// TIA Portal V20 program export: 1 tag tables, 0 data types, 2 data blocks, 4 code blocks (in call order from the OBs), 4 instance data blocks

VAR_GLOBAL   // PLC tag table "默认变量表"
   右顶升V90_Drive_IN AT %I68.0 : "PD_TEL3_IN";
   右顶升V90_Drive_OUT AT %Q68.0 : "PD_TEL3_OUT";
   左顶升IS620F_Drive_IN AT %I86.0 : "PD_TEL3_IN";
   左顶升IS620F_Drive_OUT AT %Q78.0 : "PD_TEL3_OUT";
   System_Byte AT %MB1 : Byte;
   FirstScan AT %M1.0 : Bool;
   DiagStatusUpdate AT %M1.1 : Bool;
   AlwaysTRUE AT %M1.2 : Bool;
   AlwaysFALSE AT %M1.3 : Bool;
   Clock_Byte AT %MB0 : Byte;
   Clock_10Hz AT %M0.0 : Bool;
   Clock_5Hz AT %M0.1 : Bool;
   "Clock_2.5Hz" AT %M0.2 : Bool;
   Clock_2Hz AT %M0.3 : Bool;
   "Clock_1.25Hz" AT %M0.4 : Bool;
   Clock_1Hz AT %M0.5 : Bool;
   "Clock_0.625Hz" AT %M0.6 : Bool;
   "Clock_0.5Hz" AT %M0.7 : Bool;
   右顶升V90控制字 AT %MW2 : Word;
   左顶升IS620F控制字 AT %MW4 : Word;
   左_回原模式 AT %MW6 : Int;
   左_绝对位置 AT %MD8 : Real;
   左_绝对速度 AT %MD12 : Real;
   左_相对位置 AT %MD16 : Real;
   左_相对速度 AT %MD20 : Real;
   左_点动速度 AT %MD24 : Real;
   左顶升IS620F状态字 AT %MW28 : Word;
   左顶升当前位置 AT %MD30 : Real;
   左顶升当前速度 AT %MD34 : Real;
   右顶升V90状态字 AT %MW38 : Word;
   右_回原模式 AT %MW40 : Int;
   右_绝对位置 AT %MD42 : Real;
   右_绝对速度 AT %MD46 : Real;
   右_相对位置 AT %MD50 : Real;
   右_相对速度 AT %MD54 : Real;
   右_点动速度 AT %MD58 : Real;
   右顶升当前位置 AT %MD62 : Real;
   右顶升当前速度 AT %MD66 : Real;
END_VAR

DATA_BLOCK "1200_上传"   // DB2
{ S7_Optimized_Access := 'FALSE' }
   VAR
      位1 : Bool;
      位2 : Bool;
      位3 : Bool;
      位4 : Bool;
      位5 : Bool;
      位6 : Bool;
      位7 : Bool;
      位8 : Bool;
      位9 : Bool;
      位10 : Bool;
      位11 : Bool;
      位12 : Bool;
      位13 : Bool;
      位14 : Bool;
      位15 : Bool;
      位16 : Bool;
      位17 : Bool;
      位18 : Bool;
      位19 : Bool;
      位20 : Bool;
      位21 : Bool;
      位22 : Bool;
      位23 : Bool;
      位24 : Bool;
      位25 : Bool;
      位26 : Bool;
      位27 : Bool;
      位28 : Bool;
      位29 : Bool;
      位30 : Bool;
      整型1 : Int;
      整型2 : Int;
      整型3 : Int;
      整型4 : Int;
      整型5 : Int;
      整型6 : Int;
      整型7 : Int;
      整型8 : Int;
      整型9 : Int;
      整型10 : Int;
      浮点数1 : Real;
      浮点数2 : Real;
      浮点数3 : Real;
      浮点数4 : Real;
      浮点数5 : Real;
      浮点数6 : Real;
      浮点数7 : Real;
      浮点数8 : Real;
      浮点数9 : Real;
      浮点数10 : Real;
      浮点数11 : Real;
      浮点数12 : Real;
      浮点数13 : Real;
      浮点数14 : Real;
      浮点数15 : Real;
      浮点数16 : Real;
      浮点数17 : Real;
      浮点数18 : Real;
      浮点数19 : Real;
   END_VAR
BEGIN
END_DATA_BLOCK

DATA_BLOCK "1200_下载"   // DB1
{ S7_Optimized_Access := 'FALSE' }
   VAR
      位1 : Bool;
      位2 : Bool;
      位3 : Bool;
      位4 : Bool;
      位5 : Bool;
      位6 : Bool;
      位7 : Bool;
      位8 : Bool;
      位9 : Bool;
      位10 : Bool;
      位11 : Bool;
      位12 : Bool;
      位13 : Bool;
      位14 : Bool;
      位15 : Bool;
      位16 : Bool;
      位17 : Bool;
      位18 : Bool;
      位19 : Bool;
      位20 : Bool;
      位21 : Bool;
      位22 : Bool;
      位23 : Bool;
      位24 : Bool;
      位25 : Bool;
      位26 : Bool;
      位27 : Bool;
      位28 : Bool;
      位29 : Bool;
      位30 : Bool;
      整型1 : Int;
      整型2 : Int;
      整型3 : Int;
      整型4 : Int;
      整型5 : Int;
      整型6 : Int;
      整型7 : Int;
      整型8 : Int;
      整型9 : Int;
      整型10 : Int;
      浮点数1 : Real;
      浮点数2 : Real;
      浮点数3 : Real;
      浮点数4 : Real;
      浮点数5 : Real;
      浮点数6 : Real;
      浮点数7 : Real;
      浮点数8 : Real;
      浮点数9 : Real;
      浮点数10 : Real;
      浮点数11 : Real;
      浮点数12 : Real;
      浮点数13 : Real;
      浮点数14 : Real;
      浮点数15 : Real;
      浮点数16 : Real;
      浮点数17 : Real;
      浮点数18 : Real;
      浮点数19 : Real;
   END_VAR
BEGIN
END_DATA_BLOCK

ORGANIZATION_BLOCK "Main"   // OB1, LAD, ProgramCycle
TITLE = "Main Program Sweep (Cycle)"
{ S7_Optimized_Access := 'TRUE' }
// stored: SetENOAutomatically false
   VAR_INPUT
      Initial_Call : Bool;   // Initial call of this OB
      Remanence : Bool;   // =True, if remanent data are available
   END_VAR
   VAR_TEMP
      done : Bool;
      erro : Bool;
      cuowuma : Word;
   END_VAR
BEGIN
END_ORGANIZATION_BLOCK

FUNCTION_BLOCK "定位轴基本控制"   // FB1, LAD
{ S7_Optimized_Access := 'TRUE' }
// stored: MemoryReserve 100, SetENOAutomatically false
   VAR_INPUT
      轴号 : TO_PositioningAxis;
      使能 : Bool;
      回原 : Bool;
      回原模式 : Int;
      绝对定位 : Bool;
      相对定位 : Bool;
      暂停 : Bool;
      复位 : Bool;
      绝对位置 : Real;
      绝对速度 : Real;
      相对位置 : Real;
      相对速度 : Real;
      点动正转 : Bool;
      点动反转 : Bool;
      点动速度 : Real;
   END_VAR
   VAR_OUTPUT
      轴已启用 : Bool;
      使能错误 : Bool;
      回原完成 : Bool;
      回原错误 : Bool;
      绝对定位完成 : Bool;
      绝对定位错误 : Bool;
      相对定位完成 : Bool;
      相对定位错误 : Bool;
      点动中 : Bool;
      点动错误 : Bool;
      当前位置 : Real;
      当前速度 : Real;
   END_VAR
   VAR
      MC_Power_Instance { S7_SetPoint := 'True'} : MC_Power;
      MC_Home_Instance { S7_SetPoint := 'True'} : MC_Home;
      MC_MoveAbsolute_Instance { S7_SetPoint := 'True'} : MC_MoveAbsolute;
      MC_MoveRelative_Instance { S7_SetPoint := 'True'} : MC_MoveRelative;
      MC_Reset_Instance { S7_SetPoint := 'True'} : MC_Reset;
      MC_Halt_Instance { S7_SetPoint := 'True'} : MC_Halt;
      MC_MoveJog_Instance { S7_SetPoint := 'True'} : MC_MoveJog;
   END_VAR
   VAR_TEMP
      复位完成 : Bool;
      复位错误 : Bool;
      暂停完成 : Bool;
      暂停错误 : Bool;
   END_VAR
   VAR_TEMP   // added for the SCL form of the ladder/FBD networks
      _w1 : Bool;
      _w2 : Bool;
      _w3 : Bool;
   END_VAR
BEGIN

REGION Network 1
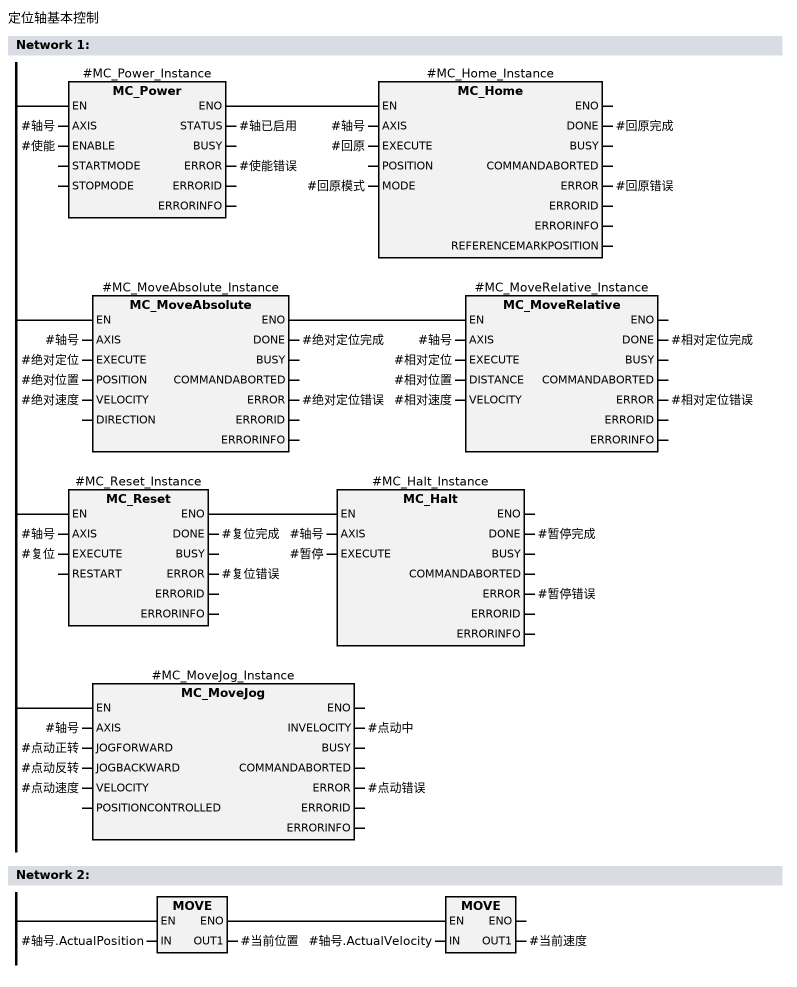
   RUNG wire#powerrail
      #MC_Power_Instance.MC_Power(Axis := #轴号, Enable := #使能, StartMode :=, StopMode :=, Status => #轴已启用, Busy =>, Error => #使能错误, ErrorID =>, ErrorInfo =>)
      #MC_Home_Instance.MC_Home(Axis := #轴号, Execute := #回原, Position :=, Mode := #回原模式, Done => #回原完成, Busy =>, CommandAborted =>, Error => #回原错误, ErrorID =>, ErrorInfo =>, ReferenceMarkPosition =>)
   END_RUNG
   RUNG wire#powerrail
      #MC_MoveAbsolute_Instance.MC_MoveAbsolute(Axis := #轴号, Execute := #绝对定位, Position := #绝对位置, Velocity := #绝对速度, Direction :=, Done => #绝对定位完成, Busy =>, CommandAborted =>, Error => #绝对定位错误, ErrorID =>, ErrorInfo =>)
      #MC_MoveRelative_Instance.MC_MoveRelative(Axis := #轴号, Execute := #相对定位, Distance := #相对位置, Velocity := #相对速度, Done => #相对定位完成, Busy =>, CommandAborted =>, Error => #相对定位错误, ErrorID =>, ErrorInfo =>)
   END_RUNG
   RUNG wire#powerrail
      #MC_Reset_Instance.MC_Reset(Axis := #轴号, Execute := #复位, Restart :=, Done => #复位完成, Busy =>, Error => #复位错误, ErrorID =>, ErrorInfo =>)
      #MC_Halt_Instance.MC_Halt(Axis := #轴号, Execute := #暂停, Done => #暂停完成, Busy =>, CommandAborted =>, Error => #暂停错误, ErrorID =>, ErrorInfo =>)
   END_RUNG
   RUNG wire#powerrail
      #MC_MoveJog_Instance.MC_MoveJog(Axis := #轴号, JogForward := #点动正转, JogBackward := #点动反转, Velocity := #点动速度, PositionControlled :=, InVelocity => #点动中, Busy =>, CommandAborted =>, Error => #点动错误, ErrorID =>, ErrorInfo =>)
   END_RUNG
   // the same network as SCL:
   #MC_Power_Instance(Axis := #轴号, Enable := #使能, Status => #轴已启用, Error => #使能错误, ENO => #_w1);   // MC_Power
   IF #_w1 THEN
       #MC_Home_Instance(Axis := #轴号, Execute := #回原, Mode := #回原模式, Done => #回原完成, Error => #回原错误);   // MC_Home
   END_IF;
   #MC_MoveAbsolute_Instance(Axis := #轴号,   // MC_MoveAbsolute
                           Execute := #绝对定位,
                           Position := #绝对位置,
                           Velocity := #绝对速度,
                           Done => #绝对定位完成,
                           Error => #绝对定位错误,
                           ENO => #_w2);
   IF #_w2 THEN
       #MC_MoveRelative_Instance(Axis := #轴号,   // MC_MoveRelative
                               Execute := #相对定位,
                               Distance := #相对位置,
                               Velocity := #相对速度,
                               Done => #相对定位完成,
                               Error => #相对定位错误);
   END_IF;
   #MC_Reset_Instance(Axis := #轴号, Execute := #复位, Done => #复位完成, Error => #复位错误, ENO => #_w3);   // MC_Reset
   IF #_w3 THEN
       #MC_Halt_Instance(Axis := #轴号, Execute := #暂停, Done => #暂停完成, Error => #暂停错误);   // MC_Halt
   END_IF;
   #MC_MoveJog_Instance(Axis := #轴号,   // MC_MoveJog
                        JogForward := #点动正转,
                        JogBackward := #点动反转,
                        Velocity := #点动速度,
                        InVelocity => #点动中,
                        Error => #点动错误);
END_REGION

REGION Network 2
   RUNG wire#powerrail
      Move(in := #轴号.ActualPosition, out1 => #当前位置)
      Move(in := #轴号.ActualVelocity, out1 => #当前速度)
   END_RUNG
   // the same network as SCL:
   #当前位置 := #轴号.ActualPosition;
   #当前速度 := #轴号.ActualVelocity;
END_REGION
END_FUNCTION_BLOCK

FUNCTION "右顶升伺服" : Void   // FC2, LAD
{ S7_Optimized_Access := 'TRUE' }
// stored: SetENOAutomatically false
BEGIN

REGION Network 1 (SCL)
   "右顶升V90控制字".%X0 := "1200_下载".位9;
   "右顶升V90控制字".%X1 := "1200_下载".位10;
   "右顶升V90控制字".%X2 := "1200_下载".位11;
   "右顶升V90控制字".%X3 := "1200_下载".位12;
   "右顶升V90控制字".%X4 := "1200_下载".位13;
   "右顶升V90控制字".%X5 := "1200_下载".位14;
   "右顶升V90控制字".%X6 := "1200_下载".位15;
   "右顶升V90控制字".%X7 := "1200_下载".位16;

   "右_回原模式" := "1200_下载".整型2;

   "右_绝对位置" := "1200_下载".浮点数6;
   "右_绝对速度" := "1200_下载".浮点数7;
   "右_相对位置" := "1200_下载".浮点数8;
   "右_相对速度" := "1200_下载".浮点数9;
   "右_点动速度" := "1200_下载".浮点数10;
END_REGION

REGION Network 2
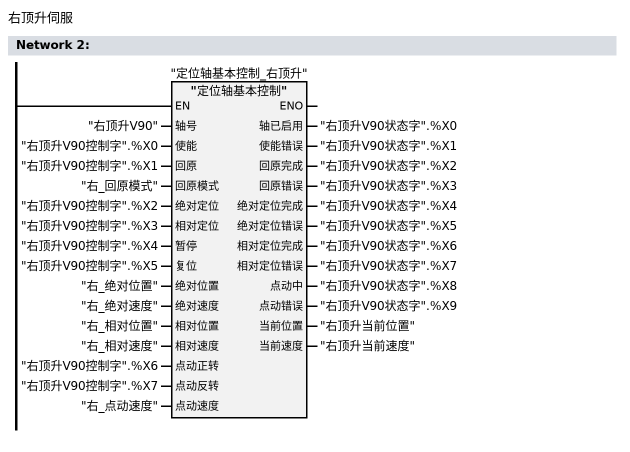
   RUNG wire#powerrail
      "定位轴基本控制_右顶升"(轴号 := "右顶升V90", 使能 := "右顶升V90控制字".%X0, 回原 := "右顶升V90控制字".%X1, 回原模式 := "右_回原模式", 绝对定位 := "右顶升V90控制字".%X2, 相对定位 := "右顶升V90控制字".%X3, 暂停 := "右顶升V90控制字".%X4, 复位 := "右顶升V90控制字".%X5, 绝对位置 := "右_绝对位置", 绝对速度 := "右_绝对速度", 相对位置 := "右_相对位置", 相对速度 := "右_相对速度", 点动正转 := "右顶升V90控制字".%X6, 点动反转 := "右顶升V90控制字".%X7, 点动速度 := "右_点动速度", 轴已启用 => "右顶升V90状态字".%X0, 使能错误 => "右顶升V90状态字".%X1, 回原完成 => "右顶升V90状态字".%X2, 回原错误 => "右顶升V90状态字".%X3, 绝对定位完成 => "右顶升V90状态字".%X4, 绝对定位错误 => "右顶升V90状态字".%X5, 相对定位完成 => "右顶升V90状态字".%X6, 相对定位错误 => "右顶升V90状态字".%X7, 点动中 => "右顶升V90状态字".%X8, 点动错误 => "右顶升V90状态字".%X9, 当前位置 => "右顶升当前位置", 当前速度 => "右顶升当前速度")
   END_RUNG
   // the same network as SCL:
   "定位轴基本控制_右顶升"(轴号 := "右顶升V90",   // "定位轴基本控制"
                 使能 := "右顶升V90控制字".%X0,
                 回原 := "右顶升V90控制字".%X1,
                 回原模式 := "右_回原模式",
                 绝对定位 := "右顶升V90控制字".%X2,
                 相对定位 := "右顶升V90控制字".%X3,
                 暂停 := "右顶升V90控制字".%X4,
                 复位 := "右顶升V90控制字".%X5,
                 绝对位置 := "右_绝对位置",
                 绝对速度 := "右_绝对速度",
                 相对位置 := "右_相对位置",
                 相对速度 := "右_相对速度",
                 点动正转 := "右顶升V90控制字".%X6,
                 点动反转 := "右顶升V90控制字".%X7,
                 点动速度 := "右_点动速度",
                 轴已启用 => "右顶升V90状态字".%X0,
                 使能错误 => "右顶升V90状态字".%X1,
                 回原完成 => "右顶升V90状态字".%X2,
                 回原错误 => "右顶升V90状态字".%X3,
                 绝对定位完成 => "右顶升V90状态字".%X4,
                 绝对定位错误 => "右顶升V90状态字".%X5,
                 相对定位完成 => "右顶升V90状态字".%X6,
                 相对定位错误 => "右顶升V90状态字".%X7,
                 点动中 => "右顶升V90状态字".%X8,
                 点动错误 => "右顶升V90状态字".%X9,
                 当前位置 => "右顶升当前位置",
                 当前速度 => "右顶升当前速度");
END_REGION

REGION Network 3 (SCL)
   "1200_上传".位11 := "右顶升V90状态字".%X0;
   "1200_上传".位12 := "右顶升V90状态字".%X1;
   "1200_上传".位13 := "右顶升V90状态字".%X2;
   "1200_上传".位14 := "右顶升V90状态字".%X3;
   "1200_上传".位15 := "右顶升V90状态字".%X4;
   "1200_上传".位16 := "右顶升V90状态字".%X5;
   "1200_上传".位17 := "右顶升V90状态字".%X6;
   "1200_上传".位18 := "右顶升V90状态字".%X7;
   "1200_上传".位19 := "右顶升V90状态字".%X8;
   "1200_上传".位20 := "右顶升V90状态字".%X9;

   "1200_上传".浮点数3 := "右顶升当前位置";
   "1200_上传".浮点数4 := "右顶升当前速度";
END_REGION
END_FUNCTION

FUNCTION "左顶升伺服" : Void   // FC1, LAD
{ S7_Optimized_Access := 'TRUE' }
// stored: SetENOAutomatically false
BEGIN

REGION Network 1 (SCL)
   "左顶升IS620F控制字".%X0 := "1200_下载".位1;
   "左顶升IS620F控制字".%X1 := "1200_下载".位2;
   "左顶升IS620F控制字".%X2 := "1200_下载".位3;
   "左顶升IS620F控制字".%X3 := "1200_下载".位4;
   "左顶升IS620F控制字".%X4 := "1200_下载".位5;
   "左顶升IS620F控制字".%X5 := "1200_下载".位6;
   "左顶升IS620F控制字".%X6 := "1200_下载".位7;
   "左顶升IS620F控制字".%X7 := "1200_下载".位8;

   "左_回原模式" := "1200_下载".整型1;

   "左_绝对位置" := "1200_下载".浮点数1;
   "左_绝对速度" := "1200_下载".浮点数2;
   "左_相对位置" := "1200_下载".浮点数3;
   "左_相对速度" := "1200_下载".浮点数4;
   "左_点动速度" := "1200_下载".浮点数5;
END_REGION

REGION Network 2
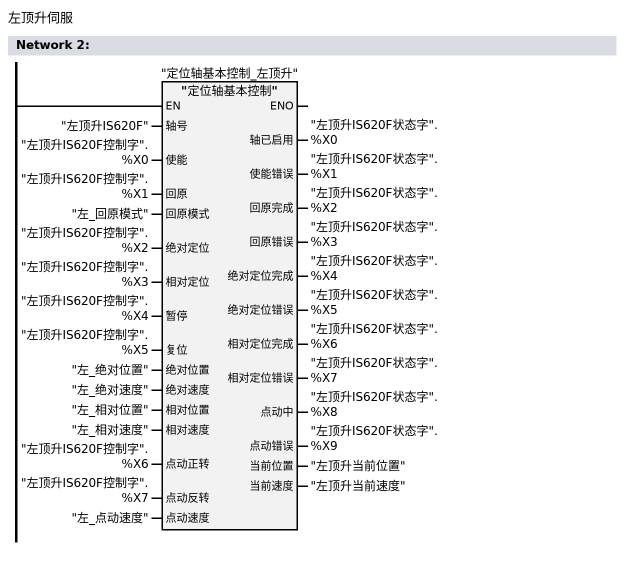
   RUNG wire#powerrail
      "定位轴基本控制_左顶升"(轴号 := "左顶升IS620F", 使能 := "左顶升IS620F控制字".%X0, 回原 := "左顶升IS620F控制字".%X1, 回原模式 := "左_回原模式", 绝对定位 := "左顶升IS620F控制字".%X2, 相对定位 := "左顶升IS620F控制字".%X3, 暂停 := "左顶升IS620F控制字".%X4, 复位 := "左顶升IS620F控制字".%X5, 绝对位置 := "左_绝对位置", 绝对速度 := "左_绝对速度", 相对位置 := "左_相对位置", 相对速度 := "左_相对速度", 点动正转 := "左顶升IS620F控制字".%X6, 点动反转 := "左顶升IS620F控制字".%X7, 点动速度 := "左_点动速度", 轴已启用 => "左顶升IS620F状态字".%X0, 使能错误 => "左顶升IS620F状态字".%X1, 回原完成 => "左顶升IS620F状态字".%X2, 回原错误 => "左顶升IS620F状态字".%X3, 绝对定位完成 => "左顶升IS620F状态字".%X4, 绝对定位错误 => "左顶升IS620F状态字".%X5, 相对定位完成 => "左顶升IS620F状态字".%X6, 相对定位错误 => "左顶升IS620F状态字".%X7, 点动中 => "左顶升IS620F状态字".%X8, 点动错误 => "左顶升IS620F状态字".%X9, 当前位置 => "左顶升当前位置", 当前速度 => "左顶升当前速度")
   END_RUNG
   // the same network as SCL:
   "定位轴基本控制_左顶升"(轴号 := "左顶升IS620F",   // "定位轴基本控制"
                 使能 := "左顶升IS620F控制字".%X0,
                 回原 := "左顶升IS620F控制字".%X1,
                 回原模式 := "左_回原模式",
                 绝对定位 := "左顶升IS620F控制字".%X2,
                 相对定位 := "左顶升IS620F控制字".%X3,
                 暂停 := "左顶升IS620F控制字".%X4,
                 复位 := "左顶升IS620F控制字".%X5,
                 绝对位置 := "左_绝对位置",
                 绝对速度 := "左_绝对速度",
                 相对位置 := "左_相对位置",
                 相对速度 := "左_相对速度",
                 点动正转 := "左顶升IS620F控制字".%X6,
                 点动反转 := "左顶升IS620F控制字".%X7,
                 点动速度 := "左_点动速度",
                 轴已启用 => "左顶升IS620F状态字".%X0,
                 使能错误 => "左顶升IS620F状态字".%X1,
                 回原完成 => "左顶升IS620F状态字".%X2,
                 回原错误 => "左顶升IS620F状态字".%X3,
                 绝对定位完成 => "左顶升IS620F状态字".%X4,
                 绝对定位错误 => "左顶升IS620F状态字".%X5,
                 相对定位完成 => "左顶升IS620F状态字".%X6,
                 相对定位错误 => "左顶升IS620F状态字".%X7,
                 点动中 => "左顶升IS620F状态字".%X8,
                 点动错误 => "左顶升IS620F状态字".%X9,
                 当前位置 => "左顶升当前位置",
                 当前速度 => "左顶升当前速度");
END_REGION

REGION Network 3 (SCL)
   "1200_上传".位1 := "左顶升IS620F状态字".%X0;
   "1200_上传".位2 := "左顶升IS620F状态字".%X1;
   "1200_上传".位3 := "左顶升IS620F状态字".%X2;
   "1200_上传".位4 := "左顶升IS620F状态字".%X3;
   "1200_上传".位5 := "左顶升IS620F状态字".%X4;
   "1200_上传".位6 := "左顶升IS620F状态字".%X5;
   "1200_上传".位7 := "左顶升IS620F状态字".%X6;
   "1200_上传".位8 := "左顶升IS620F状态字".%X7;
   "1200_上传".位9 := "左顶升IS620F状态字".%X8;
   "1200_上传".位10 := "左顶升IS620F状态字".%X9;

   "1200_上传".浮点数1 := "左顶升当前位置";
   "1200_上传".浮点数2 := "左顶升当前速度";
END_REGION
END_FUNCTION

DATA_BLOCK "定位轴基本控制_右顶升"   // DB6
// stored: InstanceOfName 定位轴基本控制, InstanceOfType FB
"定位轴基本控制"
BEGIN
END_DATA_BLOCK

DATA_BLOCK "定位轴基本控制_左顶升"   // DB5
// stored: InstanceOfName 定位轴基本控制, InstanceOfType FB
"定位轴基本控制"
BEGIN
END_DATA_BLOCK

DATA_BLOCK "右顶升V90"   // DB3, Motion_DB
AUTHOR : SIMATIC
FAMILY : BasicMC
NAME : TO_PosAx
VERSION : 8.0
// stored: InstanceOfName TO_PositioningAxis, OfSystemLibElement TO_PositioningAxis, OfSystemLibVersion 8.0
TO_PositioningAxis   // technology object, version 8.0
   // // inherited from TO_SpeedAxis
   // // inherited from TO_Axis
   // // inherited from TO_AnyMotionObject
   // VAR
   //    Header : TO_Struct_Header;
   // END_VAR
   // VAR
   //    Position { ExternalWritable := 'False'} : Real;
   //    Velocity { ExternalWritable := 'False'} : Real;
   //    ActualPosition { ExternalWritable := 'False'} : Real;
   //    ActualVelocity { ExternalWritable := 'False'} : Real;
   //    Actor { S7_SetPoint := 'True'} : TO_Struct_Actor;
   //    Sensor { S7_SetPoint := 'True'} : Array[1..1] of TO_Struct_Sensor;
   //    Units { ExternalWritable := 'False'; S7_SetPoint := 'True'} : TO_Struct_Units;
   //    Mechanics { ExternalWritable := 'False'; S7_SetPoint := 'True'} : TO_Struct_Mechanics;
   //    DynamicLimits { ExternalWritable := 'False'; S7_SetPoint := 'True'} : TO_Struct_DynamicLimits;
   //    DynamicDefaults { S7_SetPoint := 'True'} : TO_Struct_DynamicDefaults;
   //    Modulo { ExternalWritable := 'False'; S7_SetPoint := 'True'} : TO_Struct_Modulo;
   //    PositionLimits_SW { S7_SetPoint := 'True'} : TO_Struct_PositionLimitsSW;
   //    PositionLimits_HW { S7_SetPoint := 'True'} : TO_Struct_PositionLimitsHW;
   //    Homing { S7_SetPoint := 'True'} : TO_Struct_Homing;
   //    PositionControl { ExternalWritable := 'False'; S7_SetPoint := 'True'} : TO_Struct_PositionControl;
   //    FollowingError { ExternalWritable := 'False'; S7_SetPoint := 'True'} : TO_Struct_FollowingError;
   //    PositioningMonitoring { ExternalWritable := 'False'; S7_SetPoint := 'True'} : TO_Struct_PositioningMonitoring;
   //    StandstillSignal { ExternalWritable := 'False'; S7_SetPoint := 'True'} : TO_Struct_StandstillSignal;
   //    Simulation { ExternalWritable := 'False'; S7_SetPoint := 'True'} : TO_Struct_Simulation;
   //    StatusPositioning { ExternalWritable := 'False'; S7_SetPoint := 'True'} : TO_Struct_StatusPositioning;
   //    StatusDrive { ExternalWritable := 'False'; S7_SetPoint := 'True'} : TO_Struct_StatusDrive;
   //    StatusSensor { ExternalWritable := 'False'; S7_SetPoint := 'True'} : Array[1..1] of TO_Struct_StatusSensor;
   //    StatusBits { ExternalWritable := 'False'; S7_SetPoint := 'True'} : TO_Struct_StatusBits;
   //    ErrorBits { ExternalWritable := 'False'; S7_SetPoint := 'True'} : TO_Struct_ErrorBits;
   //    ControlPanel { S7_SetPoint := 'True'} : TO_Struct_ControlPanel;
   //    Internal { S7_SetPoint := 'True'} : Array[1..4] of TO_Struct_Internal;
   // END_VAR
BEGIN
   Header.VersionMaj := 8;
   Header.VersionMin := 0;
   Header."Type" := 1;
   Actor."Type" := 1;
   Actor.DataAdaption := 1;
   Actor.Interface.AddressIn.RID := 16#0208_070C;
   Actor.Interface.AddressIn.AREA := 16#81;
   Actor.Interface.AddressIn.OFFSET := 544;
   Actor.Interface.AddressOut.RID := 16#0208_070D;
   Actor.Interface.AddressOut.AREA := 16#82;
   Actor.Interface.AddressOut.OFFSET := 544;
   Sensor[1].DataAdaption := 1;
   Sensor[1].Interface.AddressIn.RID := 16#0208_070C;
   Sensor[1].Interface.AddressIn.AREA := 16#81;
   Sensor[1].Interface.AddressIn.OFFSET := 544;
   Sensor[1].Interface.AddressOut.RID := 16#0208_070D;
   Sensor[1].Interface.AddressOut.AREA := 16#82;
   Sensor[1].Interface.AddressOut.OFFSET := 544;
   Sensor[1].Interface."Type" := 2;
   DynamicLimits.MinVelocity := 0.0;
   DynamicDefaults.Acceleration := 50.0;
   DynamicDefaults.Deceleration := 50.0;
   DynamicDefaults.EmergencyDeceleration := 125.0;
   _Sensor[1].Interface.EncoderConnection := 7;
END_DATA_BLOCK

DATA_BLOCK "左顶升IS620F"   // DB4, Motion_DB
AUTHOR : SIMATIC
FAMILY : BasicMC
NAME : TO_PosAx
VERSION : 8.0
// stored: InstanceOfName TO_PositioningAxis, OfSystemLibElement TO_PositioningAxis, OfSystemLibVersion 8.0
TO_PositioningAxis   // technology object, version 8.0
   // // inherited from TO_SpeedAxis
   // // inherited from TO_Axis
   // // inherited from TO_AnyMotionObject
   // VAR
   //    Header : TO_Struct_Header;
   // END_VAR
   // VAR
   //    Position { ExternalWritable := 'False'} : Real;
   //    Velocity { ExternalWritable := 'False'} : Real;
   //    ActualPosition { ExternalWritable := 'False'} : Real;
   //    ActualVelocity { ExternalWritable := 'False'} : Real;
   //    Actor { S7_SetPoint := 'True'} : TO_Struct_Actor;
   //    Sensor { S7_SetPoint := 'True'} : Array[1..1] of TO_Struct_Sensor;
   //    Units { ExternalWritable := 'False'; S7_SetPoint := 'True'} : TO_Struct_Units;
   //    Mechanics { ExternalWritable := 'False'; S7_SetPoint := 'True'} : TO_Struct_Mechanics;
   //    DynamicLimits { ExternalWritable := 'False'; S7_SetPoint := 'True'} : TO_Struct_DynamicLimits;
   //    DynamicDefaults { S7_SetPoint := 'True'} : TO_Struct_DynamicDefaults;
   //    Modulo { ExternalWritable := 'False'; S7_SetPoint := 'True'} : TO_Struct_Modulo;
   //    PositionLimits_SW { S7_SetPoint := 'True'} : TO_Struct_PositionLimitsSW;
   //    PositionLimits_HW { S7_SetPoint := 'True'} : TO_Struct_PositionLimitsHW;
   //    Homing { S7_SetPoint := 'True'} : TO_Struct_Homing;
   //    PositionControl { ExternalWritable := 'False'; S7_SetPoint := 'True'} : TO_Struct_PositionControl;
   //    FollowingError { ExternalWritable := 'False'; S7_SetPoint := 'True'} : TO_Struct_FollowingError;
   //    PositioningMonitoring { ExternalWritable := 'False'; S7_SetPoint := 'True'} : TO_Struct_PositioningMonitoring;
   //    StandstillSignal { ExternalWritable := 'False'; S7_SetPoint := 'True'} : TO_Struct_StandstillSignal;
   //    Simulation { ExternalWritable := 'False'; S7_SetPoint := 'True'} : TO_Struct_Simulation;
   //    StatusPositioning { ExternalWritable := 'False'; S7_SetPoint := 'True'} : TO_Struct_StatusPositioning;
   //    StatusDrive { ExternalWritable := 'False'; S7_SetPoint := 'True'} : TO_Struct_StatusDrive;
   //    StatusSensor { ExternalWritable := 'False'; S7_SetPoint := 'True'} : Array[1..1] of TO_Struct_StatusSensor;
   //    StatusBits { ExternalWritable := 'False'; S7_SetPoint := 'True'} : TO_Struct_StatusBits;
   //    ErrorBits { ExternalWritable := 'False'; S7_SetPoint := 'True'} : TO_Struct_ErrorBits;
   //    ControlPanel { S7_SetPoint := 'True'} : TO_Struct_ControlPanel;
   //    Internal { S7_SetPoint := 'True'} : Array[1..4] of TO_Struct_Internal;
   // END_VAR
BEGIN
   Header.VersionMaj := 8;
   Header.VersionMin := 0;
   Header."Type" := 1;
   Actor."Type" := 1;
   Actor.DataAdaption := 1;
   Actor.Interface.AddressIn.RID := 16#0208_070C;
   Actor.Interface.AddressIn.AREA := 16#81;
   Actor.Interface.AddressIn.OFFSET := 688;
   Actor.Interface.AddressOut.RID := 16#0208_070D;
   Actor.Interface.AddressOut.AREA := 16#82;
   Actor.Interface.AddressOut.OFFSET := 624;
   Sensor[1].DataAdaption := 1;
   Sensor[1].Interface.AddressIn.RID := 16#0208_070C;
   Sensor[1].Interface.AddressIn.AREA := 16#81;
   Sensor[1].Interface.AddressIn.OFFSET := 688;
   Sensor[1].Interface.AddressOut.RID := 16#0208_070D;
   Sensor[1].Interface.AddressOut.AREA := 16#82;
   Sensor[1].Interface.AddressOut.OFFSET := 624;
   Sensor[1].Interface."Type" := 2;
   DynamicLimits.MinVelocity := 0.0;
   DynamicDefaults.Acceleration := 50.0;
   DynamicDefaults.Deceleration := 50.0;
   DynamicDefaults.EmergencyDeceleration := 125.0;
   _Sensor[1].Interface.EncoderConnection := 7;
END_DATA_BLOCK
